TYPE PM_others :
STRUCT
	power_inConv	:BOOL;
	contactor_inConv	: BOOL;
	power_outConv	:BOOL;
	contactor_outConv	: BOOL;	
	measuring_light_curtain_a	: ARRAY[0..16] OF BYTE;
	measuring_light_curtain_b	: ARRAY[0..16] OF BYTE;
END_STRUCT
END_TYPE

(* stored: Version 1.1.0.1, ProductVersion 3.1.4024.12
   DUT PM_others: Id {0bcb23e8-9eab-454e-973e-32b67b1ef0cb} *)
